{attribute 'linkalways'} 
{attribute 'no_explicit_call' := 'This FB is a CLASS and must be accessed using methods or properties'}
{attribute 'enable_dynamic_creation'}
FUNCTION_BLOCK Node_F_VN_EnclosingCircle EXTENDS VisionNode
VAR
    ipPointSet : _ITcVnContainer;
    aCenter : _TcVnPoint2_REAL;
    fRadius : _REAL(0.0);
    hrPrev : _HRESULT(S_OK);
	hresult : _HRESULT(S_OK);
END_VAR

METHOD PUBLIC  Clone : I_Node
VAR
	pNode : POINTER TO Node_F_VN_EnclosingCircle;
END_VAR
pNode := __NEW(Node_F_VN_EnclosingCircle);
Clone := pNode^;
END_METHOD

METHOD FB_init : BOOL
VAR_INPUT
	bInitRetains : BOOL; // if TRUE, the retain variables are initialized (warm start / cold start)
	bInCopyCode : BOOL;  // if TRUE, the instance afterwards gets moved into the copy code (online change)
END_VAR
AddInput('ipPointSet', ipPointSet);
AddInput('hrPrev', hrPrev);
AddOutput('aCenter', aCenter);
AddOutput('fRadius', fRadius);
AddOutput('hresult',hresult);
END_METHOD

METHOD PROTECTED OnExecute
hresult.Value := F_VN_EnclosingCircle(
	ipPointSet := ipPointSet.Value,
    aCenter := aCenter.Value,
    fRadius := fRadius.Value,
	hrPrev:= hrPrev.Value);
END_METHOD

METHOD PUBLIC PreExecutionCheck
VAR_INPUT
	Check : I_PreExecutionChecks;
END_VAR
Check.IsTrue(ipPointSet.IsValid, 'ipPointSet must be a valid container');
Check.IsTrue((ipPointSet.IsType(TC_GLOBAL_CONST_LIST.ContainerType_Vector_TcVnPoint2_DINT) OR
              ipPointSet.IsType(TC_GLOBAL_CONST_LIST.ContainerType_Vector_TcVnPoint2_REAL)),
              'ipPointSet contains incorrect type');
END_METHOD

END_FUNCTION_BLOCK

(* stored: Version 1.1.0.1, ProductVersion 3.1.4026.13
   POU Node_F_VN_EnclosingCircle: Id {803b1e86-cc4a-0068-0964-9320219c3d32}, SpecialFunc None
   Folder Constructor: Id {1aa47b4e-e2d3-0f1c-3948-a84706e83af3}
   Method Clone: Id {a86fb25d-19a0-06b0-2416-f3d5a37c43e6}
   Method FB_init: Id {f2cf5c5d-cb17-03dc-0434-df8af88ddf9d}
   Method OnExecute: Id {b537f03c-f639-0dab-0edc-d0eeb8698e9f}
   Method PreExecutionCheck: Id {0850b099-c64b-0a6e-13f3-9c657493d017} *)
